FUNCTION_BLOCK FB_System
VAR_INPUT
END_VAR
VAR_OUTPUT
END_VAR
VAR
	plcStart : PLC_Start;
	plcStop : PLC_Stop;
END_VAR

{attribute 'TcRpcEnable'}
METHOD startRuntime : BOOL
plcStart(
	NETID:= '', 
	PORT:= 851, 
	START:= TRUE, 
	TMOUT:= , 
	BUSY=> , 
	ERR=> , 
	ERRID=> );
	
plcStart(
	NETID:= '', 
	PORT:= 851, 
	START:= FALSE, 
	TMOUT:= , 
	BUSY=> , 
	ERR=> , 
	ERRID=> );
END_METHOD

{attribute 'TcRpcEnable'}
METHOD stopRuntime : BOOL
plcStop(
	NETID:= '', 
	PORT:= 851, 
	STOP:= TRUE, 
	TMOUT:= , 
	BUSY=> , 
	ERR=> , 
	ERRID=> );
	
plcStop(
	NETID:= '', 
	PORT:= 851, 
	STOP:= FALSE, 
	TMOUT:= , 
	BUSY=> , 
	ERR=> , 
	ERRID=> );
END_METHOD

END_FUNCTION_BLOCK

(* stored: Version 1.1.0.1, ProductVersion 3.1.4024.12
   POU FB_System: Id {3df11356-d723-40c5-bd16-325ffd1c8434}, SpecialFunc None
   Method startRuntime: Id {f1e1dfb1-a05a-46a8-95e0-a372db58dbfb}
   Method stopRuntime: Id {d85e402a-5466-4cae-a47b-6151c6e3078c} *)
